FUNCTION_BLOCK fb_MQTTSUB
VAR_INPUT	
	MqttClient : FB_IotMqttClient;
	sTopic : STRING;
END_VAR
VAR_IN_OUT	
	MessageQueue : FB_IotMqttMessageQueue;
END_VAR
VAR_OUTPUT
	sValue : STRING;
END_VAR
VAR
	Message : FB_IotMqttMessage;
END_VAR

MqttClient.Subscribe(sTopic:=sTopic, eQoS:=TcIotMqttQos.AtMostOnceDelivery);

IF MessageQueue.nQueuedMessages > 0 THEN
  
	 IF MessageQueue.Dequeue(fbMessage:=Message) THEN	
		
        IF Message.CompareTopic(sTopic:=sTopic) THEN
            Message.GetPayload(pPayload:=ADR(sValue), nPayloadSize:=SIZEOF(sValue), bSetNullTermination:=FALSE);
	 	END_IF	
		
	END_IF
END_IF

END_FUNCTION_BLOCK

(* stored: Version 1.1.0.1, ProductVersion 3.1.4024.12
   POU fb_MQTTSUB: Id {61620019-43a4-4164-9f43-e2ec99bef6e7}, SpecialFunc None *)
